Universal Robots PolyScope program: Put_into_box_UR5.urp

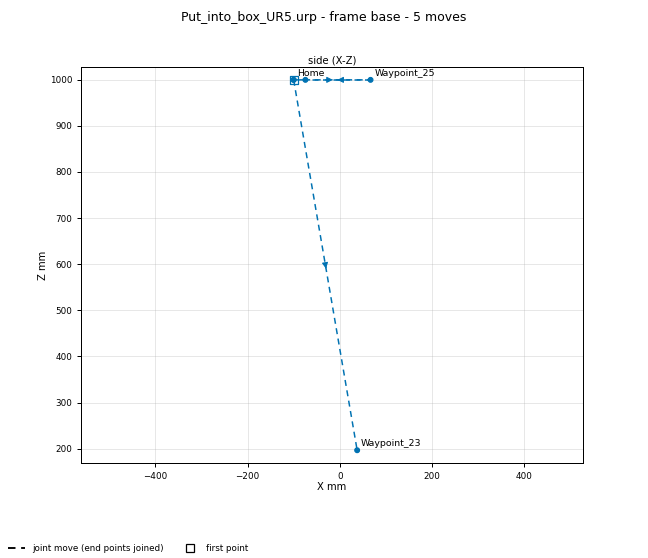
[picture p0: tool path of Put_into_box_UR5.urp in frame base, 5 of 5 moves have a stored position in this frame; points joined in program order, loops and branches not executed]
ProgramRoot directory=/programs; kinematics=(a=[0, -0.425, -0.39225, 0, 0, 0], d=[0.08916, 0, 0, 0.10915, 0.09465, 0.0823], alpha=[1.5708, 0, 0, 1.5708, -1.5708, 0], deltaTheta=[0, 0, 0, 0, 0, 0], status=notInitialized); name=Put_into_box_UR5; programVersion=(project__name=PolyScope, major__version=1, minor__version=0, svn__revision=0); robotEnvironmentFileName=default; variables=(Variable=(name=loop_1, prefersPersistentValue=false, requestANewUniqueName=false), Variable=(name=loop_2, prefersPersistentValue=false, requestANewUniqueName=false), Variable=(name=loop_3, prefersPersistentValue=false, requestANewUniqueName=false), Variable=(name=loop_4, prefersPersistentValue=false, requestANewUniqueName=false), Variable=(name=loop_5, prefersPersistentValue=false, requestANewUniqueName=false), Variable=(name=loop_6, prefersPersistentValue=false, requestANewUniqueName=false), Variable=(name=loop_7, prefersPersistentValue=false, requestANewUniqueName=false))
  MainProgram cartesianAcceleration=1.2; cartesianSpeed=0.3; jointAcceleration=1.3962634015954636; jointSpeed=1.0471975511965976; moveAsFastAsPossible=true; sharedProcessMoveBlendRadius=0.0; featureReference=(installationNameReference=Base); motionType=JOINT_SPACE; runOnlyOneCycle=true
    Action analogValue=4.0; digitalValue=0; payloadValue=0.0; selectedAnalogSensor=-1; selectedDigitalSensor=-1; setPayloadValue=true; type=NO_ACTION
    Move cartesianAcceleration=1.2; cartesianSpeed=0.3; jointAcceleration=1.3962634015954636; jointSpeed=0.17453292519943295; moveAsFastAsPossible=true; sharedProcessMoveBlendRadius=0.025; featureReference=(installationNameReference=Base); motionType=JOINT_SPACE
      Waypoint blendRadius=0.0; cartesianAcceleration=1.2; cartesianSpeed=0.3; jointAcceleration=1.3962634015954636; jointSpeed=1.0471975511965976; nextMotionTime=2.0; stoppoint=true; useSharedParameters=true; position=TCP in base x=-99.993 y=-190.994 z=999.647 mm, rx=0.0001 ry=-2.2213 rz=2.2213 rad; joints [0, -90, 0, -90, 0, 0] deg; positionType=FIXED_POSITION; name=Home
      Waypoint blendRadius=0.05; cartesianAcceleration=1.2; cartesianSpeed=0.3; jointAcceleration=1.3962634015954636; jointSpeed=1.0471975511965976; nextMotionTime=2.0; stoppoint=true; useSharedParameters=true; position=TCP in base x=66.716 y=-178.969 z=999.63 mm, rx=-0.3657 ry=2.0272 rz=-2.0272 rad; joints [20.439, -90, 0, -90, 0, 0] deg; positionType=FIXED_POSITION; name=Waypoint_25
      Popup message=Remove first bolt placed under shoulder; type=MESSAGE
      Waypoint blendRadius=0.05; cartesianAcceleration=1.2; cartesianSpeed=0.3; jointAcceleration=1.3962634015954636; jointSpeed=1.0471975511965976; nextMotionTime=2.0; stoppoint=true; useSharedParameters=true; position=TCP in base x=-74.498 y=-175.872 z=999.63 mm, rx=-0.4062 ry=-2.0012 rz=2.0011 rad; joints [-22.964, -90, 0, -90, 0, 0] deg; positionType=FIXED_POSITION; name=Waypoint_26
      Popup message=Remove second bolt placed under shoulder                                                                      Place protective pad between arm and base joint; type=MESSAGE
      Waypoint blendRadius=0.0; cartesianAcceleration=1.2; cartesianSpeed=0.3; jointAcceleration=1.3962634015954636; jointSpeed=1.0471975511965976; nextMotionTime=2.0; stoppoint=true; useSharedParameters=true; position=TCP in base x=-99.993 y=-190.994 z=999.647 mm, rx=0.0001 ry=-2.2213 rz=2.2213 rad; joints [0, -90, 0, -90, 0, 0] deg; positionType=FIXED_POSITION; name=Home
      Waypoint blendRadius=0.05; cartesianAcceleration=1.2; cartesianSpeed=0.3; jointAcceleration=1.3962634015954636; jointSpeed=1.0471975511965976; nextMotionTime=2.0; stoppoint=true; useSharedParameters=true; position=TCP in base x=37.68 y=-191.036 z=196.558 mm, rx=1.2057 ry=-1.2156 rz=1.2134 rad; joints [-0.055, 3.602, -163.716, -109.496, 0.049, 0.025] deg; positionType=FIXED_POSITION; name=Waypoint_23
      Popup message=Remove remaining bolts; type=MESSAGE
